FUNCTION MMS_TO_MMIN : LREAL
VAR_INPUT
	IN														:	LREAL;
END_VAR
VAR
END_VAR

MMS_TO_MMIN 												:= IN * 0.001 * 60;

END_FUNCTION

(* stored: Version 1.1.0.1, ProductVersion 3.1.4024.12
   POU MMS_TO_MMIN: Id {55954f0c-4287-420d-b6ab-b68be3713337}, SpecialFunc None *)
